PROGRAM AP_1
VAR
	GetPlate			:Seq_Get_Plate;
	SetPlate1			:Seq_Set_Plate_1;
	SetPlate2			:Seq_Set_Plate_2;
END_VAR

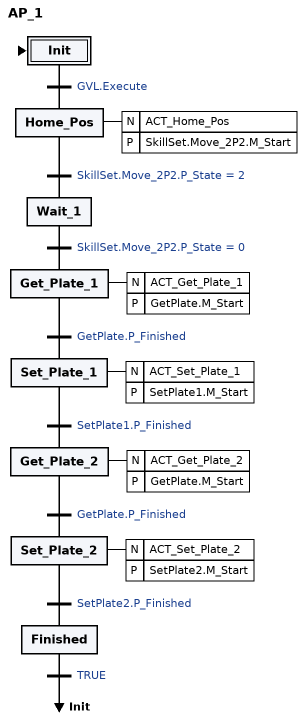
INITIAL_STEP Init:
END_STEP
TRANSITION FROM Init TO Home_Pos
    := GVL.Execute;
END_TRANSITION
STEP Home_Pos:
    ACT_Home_Pos(N);
    SkillSet.Move_2P2.M_Start(P);
END_STEP
TRANSITION FROM Home_Pos TO Wait_1
    := SkillSet.Move_2P2.P_State = 2;
END_TRANSITION
STEP Wait_1:
END_STEP
TRANSITION FROM Wait_1 TO Get_Plate_1
    := SkillSet.Move_2P2.P_State = 0;
END_TRANSITION
STEP Get_Plate_1:
    ACT_Get_Plate_1(N);
    GetPlate.M_Start(P);
END_STEP
TRANSITION FROM Get_Plate_1 TO Set_Plate_1
    := GetPlate.P_Finished;
END_TRANSITION
STEP Set_Plate_1:
    ACT_Set_Plate_1(N);
    SetPlate1.M_Start(P);
END_STEP
TRANSITION FROM Set_Plate_1 TO Get_Plate_2
    := SetPlate1.P_Finished;
END_TRANSITION
STEP Get_Plate_2:
    ACT_Get_Plate_2(N);
    GetPlate.M_Start(P);
END_STEP
TRANSITION FROM Get_Plate_2 TO Set_Plate_2
    := GetPlate.P_Finished;
END_TRANSITION
STEP Set_Plate_2:
    ACT_Set_Plate_2(N);
    SetPlate2.M_Start(P);
END_STEP
TRANSITION FROM Set_Plate_2 TO Finished
    := SetPlate2.P_Finished;
END_TRANSITION
STEP Finished:
END_STEP
TRANSITION FROM Finished TO Init
    := TRUE;
END_TRANSITION

ACTION ACT_Get_Plate_1:
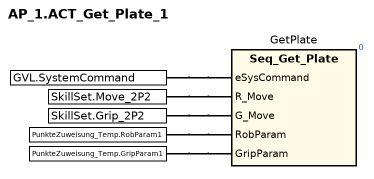
GetPlate(
    eSysCommand := GVL.SystemCommand,
    R_Move := SkillSet.Move_2P2,
    G_Move := SkillSet.Grip_2P2,
    RobParam := PunkteZuweisung_Temp.RobParam1,
    GripParam := PunkteZuweisung_Temp.GripParam1); // Seq_Get_Plate
END_ACTION

ACTION ACT_Get_Plate_2:
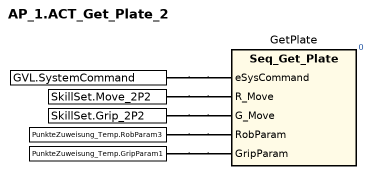
GetPlate(
    eSysCommand := GVL.SystemCommand,
    R_Move := SkillSet.Move_2P2,
    G_Move := SkillSet.Grip_2P2,
    RobParam := PunkteZuweisung_Temp.RobParam3,
    GripParam := PunkteZuweisung_Temp.GripParam1); // Seq_Get_Plate
END_ACTION

ACTION ACT_Home_Pos:
SkillSet.Move_2P2.P_RobotParam := PunkteZuweisung_Temp.PHome;
END_ACTION

ACTION ACT_Set_Plate_1:
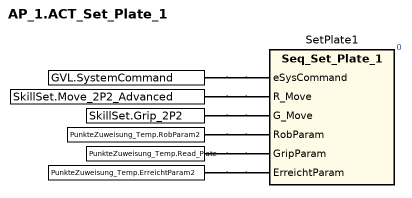
SetPlate1(
    eSysCommand := GVL.SystemCommand,
    R_Move := SkillSet.Move_2P2_Advanced,
    G_Move := SkillSet.Grip_2P2,
    RobParam := PunkteZuweisung_Temp.RobParam2,
    GripParam := PunkteZuweisung_Temp.Read_Plate,
    ErreichtParam := PunkteZuweisung_Temp.ErreichtParam2); // Seq_Set_Plate_1
END_ACTION

ACTION ACT_Set_Plate_2:
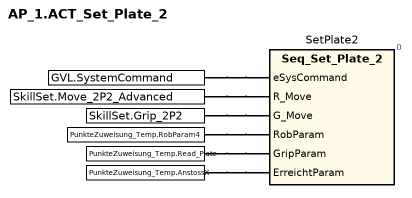
SetPlate2(
    eSysCommand := GVL.SystemCommand,
    R_Move := SkillSet.Move_2P2_Advanced,
    G_Move := SkillSet.Grip_2P2,
    RobParam := PunkteZuweisung_Temp.RobParam4,
    GripParam := PunkteZuweisung_Temp.Read_Plate,
    ErreichtParam := PunkteZuweisung_Temp.AnstossX); // Seq_Set_Plate_2
END_ACTION

END_PROGRAM

(* stored: Version 1.1.0.1
   POU AP_1: Id {3a8a7c03-4d29-456d-873b-3b80c55e380a}, SpecialFunc None
   Folder 01_Zuweisung: Id {ecd5fb79-7da5-47f5-ae11-0167aae7cac7}
   Action ACT_Get_Plate_1: Id {4c917d64-6118-40b3-9050-73e978e53fbe}
   Action ACT_Get_Plate_2: Id {4e88ce0c-50e0-40d7-b6a6-6d376a23ab12}
   Action ACT_Home_Pos: Id {c0550dcd-88e4-40a1-a94d-79534d55193d}
   Action ACT_Set_Plate_1: Id {79a81c60-47f1-474a-a8cb-80c54df6179e}
   Action ACT_Set_Plate_2: Id {97bcf6ff-9d20-4145-9151-e3784d2cb36b} *)
